// TIA Portal V17 export
// export: Created 2025-06-26T07:49:49.4526433Z, ExportSetting WithDefaults, DisplayName Totally Integrated Automation Portal, DisplayVersion V17 Update 8, DisplayName TIA Portal Openness, DisplayVersion V17 Update 8, DisplayName TIA Portal Version Control Interface, DisplayVersion V17, DisplayName STEP 7 Professional, DisplayVersion V17 Update 8, DisplayName STEP 7 Safety, DisplayVersion V17 Update 6, DisplayName WinCC Advanced, DisplayVersion V17 Update 8
FUNCTION_BLOCK "fbHysteresis"   // FB43, FBD
TITLE = Threshold detection with deadband
{ S7_Optimized_Access := 'TRUE' }
VERSION : 0.1
// stored: AutoNumber true, IsIECCheckEnabled false, IsRetainMemResEnabled false, MemoryReserve 0, SetENOAutomatically false, UDAEnableTagReadback false
   VAR_INPUT
      fValue : Real;
      fLimit : Real;
      fHysteresis : Real;
      bType : Bool;   // 0 = under the limit, 1 = over the limit
   END_VAR
   VAR_OUTPUT
      bOutput : Bool;
   END_VAR
   VAR
      State : Bool;
   END_VAR
   VAR_TEMP
      Set : Bool;
      Reset : Bool;
   END_VAR
BEGIN

REGION Network 1 (SCL)
   // Over the limit: 
   //  - output is activated when input value is greater than the limit plus half the deadband, AND STAYS ACTIVATED UNTIL the deactivation condition is reached
   //  - output is deactivated when the input value is less than the limit minus half the deadband, AND STAYS DEACTIVATED UNTIL the activation condition is reached
   // 
   // Under the limit: 
   //  - output is activated when the input value is less than the limit minus half the deadband
   //  - output is deactivated when the input value is greater than the limit plus half the deadband
   IF #bType = TRUE THEN
       #Set := #fValue > (#fLimit + #fHysteresis/2);
       #Reset := #fValue < (#fLimit - #fHysteresis/2);
   ELSE
       #Set := #fValue < (#fLimit - #fHysteresis/2);
       #Reset := #fValue > (#fLimit + #fHysteresis/2);
   END_IF;
END_REGION

REGION Network 2
   // A memory bit preserves the output state, even when the input changes. You can't have hysteresis without memory!
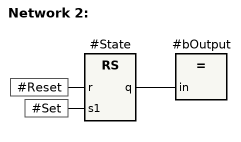
   IF #Reset THEN
       #State := FALSE;   // RS flip-flop
   END_IF;
   IF #Set THEN #State := TRUE; END_IF;
   #bOutput := #State;
END_REGION
END_FUNCTION_BLOCK
